{attribute 'linkalways'} 
{attribute 'no_explicit_call' := 'This FB is a CLASS and must be accessed using methods or properties'}
{attribute 'enable_dynamic_creation'}
FUNCTION_BLOCK ABSTRACT Alarm IMPLEMENTS I_Alarm

METHOD PUBLIC Accept
VAR_INPUT
	Visitor : I_AlarmVisitor;
END_VAR
Visitor.VisitError(this^);
END_METHOD

PROPERTY ABSTRACT Active : BOOL
GET
END_GET
END_PROPERTY

METHOD ABSTRACT Clear
END_METHOD

METHOD FB_init : BOOL
VAR_INPUT
	bInitRetains : BOOL; // if TRUE, the retain variables are initialized (warm start / cold start)
	bInCopyCode : BOOL;  // if TRUE, the instance afterwards gets moved into the copy code (online change)
	Parent : I_HostAlarms;
END_VAR
RegisterWithParent(Parent);
END_METHOD

PROPERTY ABSTRACT Message : T_MaxString
GET
END_GET
END_PROPERTY

PROPERTY ABSTRACT Reason : T_MaxString
GET
END_GET
END_PROPERTY

METHOD RegisterWithParent
VAR_INPUT
	Parent : I_HostAlarms;
END_VAR
IF Parent = 0 THEN
	RETURN;
END_IF

Parent.Alarms.AddAlarm(THIS^);
END_METHOD

METHOD PUBLIC SerializeWith
VAR_INPUT
	Serializer : I_Serializer;
END_VAR
VAR
	isActive : BOOL := Active;
	errorMessage : T_MAXSTRING := Message;
	reasonMessage : T_MAXSTRING := Reason;
END_VAR
Serializer.StartObject();
Serializer.AddKeyString('message',errorMessage);
Serializer.AddKeyBool('active',isActive);

IF reasonMessage <> '' THEN
	Serializer.AddKeyString('reason',reasonMessage);
END_IF

Serializer.EndObject();
END_METHOD

END_FUNCTION_BLOCK

(* stored: Version 1.1.0.1, ProductVersion 3.1.4024.12
   POU Alarm: Id {71bd3509-3a77-0a94-2705-a3ad83e250bc}, SpecialFunc None
   Folder Abstract: Id {0131d39e-f487-0641-11b7-adb32e39c242}
   Folder Constructor: Id {5450f8b1-7227-0795-0f4e-7c2a85062d3c}
   Method Accept: Id {354a4344-cb86-0485-1c3b-41f76fac9dc7}
   Property Active: Id {32327753-2b64-051d-2eb5-0f62f66c274d}
   Get Get: Id {02cf22be-56f7-0b63-1d1a-bdd5cdd8f6ef}
   Method Clear: Id {df360e35-c463-06e7-2ad6-0a908ff031af}
   Method FB_init: Id {172b7039-54b0-0e58-2410-0f2a4d86f948}
   Property Message: Id {58408768-0ecc-0b83-2e43-489069f7d2bc}
   Get Get: Id {7455a364-4a30-0c2a-2023-714d8beb13e9}
   Property Reason: Id {db42a7b6-e03c-0b06-1c6d-921219967bf7}
   Get Get: Id {9161ac02-8ad7-0a1e-1267-df4942b29797}
   Method RegisterWithParent: Id {50a3db7c-f4f1-0156-3933-1f93438f5c5a}
   Method SerializeWith: Id {a2ed8123-2f68-4e86-a79d-a0fb02c58153} *)
